// TwinCAT 3 PLC project Plc
// ProgramVersion: 3.1.4024.0
// libraries:
//   Tc2_Standard, * (Beckhoff Automation GmbH)
//   Tc2_System, * (Beckhoff Automation GmbH)
//   Tc2_TcpIp, * (Beckhoff Automation GmbH)
//   Tc3_Module, * (Beckhoff Automation GmbH)
//   VisuSymbols,3.5.10.0,System
// project tree:
//   Elements/Common/ E_Mode.TcDUT, ST_DigitalInput.TcDUT, ST_DigitalOutput.TcDUT, ST_ToggleCmd.TcDUT, ST_TapCmd.TcDUT
//   Elements/Lights/ E_ButtonSelection.TcDUT, FB_AnalogLamp.TcPOU, FB_DigitalLamp.TcPOU, ST_AnalogLamp_cmd.TcDUT, ST_AnalogLamp_fb.TcDUT, ST_DigitalLamp_cmd.TcDUT, ST_DigitalLamp_fb.TcDUT
//   Elements/ ST_AC_Swing.TcDUT, ST_Curtain_Status.TcDUT, ST_ACcontrol.TcDUT, ST_ACStatus.TcDUT, ST_Fan_ip.TcDUT, ST_Fan_op.TcDUT
//   / GlobalTextList.TcGTLO, PlcTask.TcTTO, Visualization Manager.TcVMO (not stored)
//   Helper/ FB_CommandHandling.TcPOU, FB_CurtainPos.TcPOU, F_Scaling.TcPOU (not stored)
//   POUs/ FB_AC.TcPOU, FB_AC_oop.TcPOU, FB_Curtain.TcPOU, FB_Dimmer.TcPOU, FB_Fan.TcPOU, FB_Lamp.TcPOU, FB_Room.TcPOU, I_AC.TcIO, MAIN.TcPOU, PRG_HallRoom.TcPOU, PRG_Kitchen.TcPOU, PRG_SmartHome.TcPOU
//   POUs/TcpIp/ FB_ACcomm.TcPOU, FB_TcpIpClient.TcPOU
//   Trials/ PRG_Testing.TcPOU
//   VISUs/ Template.TcVIS, V_Hall.TcVIS, V_House.TcVIS
// real-time tasks:
//   TASK PlcTask: cycle T#10ms, priority 20, ADS port 350
//   TASK PlcTask1: cycle T#10ms, priority 21, ADS port 351

CONFIGURATION Plc
    RESOURCE PLC ON TwinCAT3
        TASK PlcTask(INTERVAL := T#10ms, PRIORITY := 20);
        PROGRAM MAIN WITH PlcTask : MAIN;
    END_RESOURCE
END_CONFIGURATION

// ---- Elements/Common/E_Mode.TcDUT
{attribute 'qualified_only'}
{attribute 'strict'}
TYPE E_Mode :
(
	auto := 0,
	simulation := 1,
	maintenance := 2,
	manual := 3
);
END_TYPE

// ---- Elements/Common/ST_DigitalInput.TcDUT
TYPE ST_DigitalInput :
STRUCT
	hmi_In: BOOL;
	i_In AT %I* : BOOL;
	mode: E_Mode;
END_STRUCT
END_TYPE

// ---- Elements/Common/ST_DigitalOutput.TcDUT
TYPE ST_DigitalOutput :
STRUCT
	hmi_Out: BOOL;
	q_Out AT %Q* : BOOL;
	mode: E_Mode;
END_STRUCT
END_TYPE

// ---- Elements/Common/ST_ToggleCmd.TcDUT
TYPE ST_ToggleCmd :
STRUCT
	OnOff: BOOL;
END_STRUCT
END_TYPE

// ---- Elements/Common/ST_TapCmd.TcDUT
TYPE ST_TapCmd :
STRUCT
	OnOff: BOOL;
END_STRUCT
END_TYPE

// ---- Elements/Lights/E_ButtonSelection.TcDUT
{attribute 'qualified_only'}
{attribute 'strict'}
TYPE E_ButtonSelection :
(
	Tap := 0,		//	toggle if Event rising edge is detected
	Toggle := 1		//	0: off | 1: on
);
END_TYPE

// ---- Elements/Lights/ST_AnalogLamp_cmd.TcDUT
TYPE ST_AnalogLamp_cmd :
STRUCT
	OnOff: BOOL;
	brightness_SP: INT;	//SP- Setpoint
	colorCode: UDINT;
END_STRUCT
END_TYPE

// ---- Elements/Lights/ST_AnalogLamp_fb.TcDUT
TYPE ST_AnalogLamp_fb :
STRUCT
	status: BOOL;
	brightness: INT;
	colorSelected: UDINT;
	errorID: UDINT;
END_STRUCT
END_TYPE

// ---- Elements/Lights/ST_DigitalLamp_cmd.TcDUT
TYPE ST_DigitalLamp_cmd :
STRUCT
	E_ButtonSelection: E_ButtonSelection;
	Toggle: ST_ToggleCmd;
	PushButton: ST_TapCmd;
END_STRUCT
END_TYPE

// ---- Elements/Lights/ST_DigitalLamp_fb.TcDUT
TYPE ST_DigitalLamp_fb :
STRUCT
	Status: BOOL;
END_STRUCT
END_TYPE

// ---- Elements/ST_AC_Swing.TcDUT
TYPE ST_AC_Swing :
STRUCT
	HorizOn: BOOL;
	HorizOff: BOOL;
	VertiOn: BOOL;
	VertiOff: BOOL;
END_STRUCT
END_TYPE

// ---- Elements/ST_Curtain_Status.TcDUT
TYPE ST_Curtain_Status :
STRUCT
	Open	  	: BOOL;
	Close	 	: BOOL;
	OpenPerc	: INT; 	//0: Closed .. 100: Full Open	
	OpenToCloseTime: TIME := T#10S;
END_STRUCT
END_TYPE

// ---- Elements/ST_ACcontrol.TcDUT
TYPE ST_ACcontrol :
STRUCT
	OnCmd: BOOL;
	OffCmd: BOOL;
	modeSelection: INT;
	swing: ST_AC_Swing;
	tempUp: BOOL;
	tempDown: BOOL;
	tempSP: REAL;
	tempSP_prev: REAL;
END_STRUCT
END_TYPE

// ---- Elements/ST_ACStatus.TcDUT
TYPE ST_ACStatus :
STRUCT
	OnOff: BOOL;
	mode: INT;
	HorizSwingOnOff: BOOL;
	VertiSwingOnOff: BOOL;
	temp: REAL;
END_STRUCT
END_TYPE

// ---- Elements/ST_Fan_ip.TcDUT
TYPE ST_Fan_ip :
STRUCT
	OnOffCmd 	AT%I* : BOOL;
	SpeedSp		AT%I* : INT;
END_STRUCT
END_TYPE

// ---- Elements/ST_Fan_op.TcDUT
TYPE ST_Fan_op :
STRUCT
	OnOff	 	AT%Q* : BOOL;
	Speed		AT%Q* : INT;
END_STRUCT
END_TYPE

// ---- POUs/I_AC.TcIO
INTERFACE I_AC

PROPERTY AC_IPAddr : STRING
GET
END_GET
END_PROPERTY

PROPERTY ACcontrol : ST_ACcontrol
GET
END_GET
END_PROPERTY

PROPERTY ACstatus : ST_ACStatus
SET
END_SET
END_PROPERTY

END_INTERFACE

// ---- POUs/MAIN.TcPOU
PROGRAM MAIN
VAR
END_VAR


	PRG_SmartHome();
	PRG_Testing();

END_PROGRAM

// ---- POUs/PRG_SmartHome.TcPOU
PROGRAM PRG_SmartHome
VAR
	fbRoom: ARRAY[0..1] OF FB_Room;
	AC_IPAddr: STRING := '192.168.1.7';
END_VAR


	fbRoom[0](AC_IPAddr := AC_IPAddr, ACcontrol:= , ACstatus=> );
//	fbRoom[1](AC_IPAddr := );
//	PRG_HallRoom();
//	PRG_Kitchen();

END_PROGRAM

// ---- POUs/FB_Room.TcPOU
FUNCTION_BLOCK FB_Room
VAR_INPUT
	AC_IPAddr: STRING;
	ACcontrol: ST_ACcontrol;
END_VAR
VAR_OUTPUT
	ACstatus: ST_ACStatus;
END_VAR
VAR
	fbLamp : ARRAY[0..3] OF FB_Lamp;
	fbDimmer : ARRAY[0..3] OF FB_Dimmer;
	fbCurtain: FB_Curtain;
	fbAC: FB_AC;
	i: INT;
	fbAC_oop: FB_AC_oop;
END_VAR

	
	FOR i := 0 TO 3 BY 1 DO
		fbLamp[i]();
		fbDimmer[i]();
	END_FOR
	
	//fbAC(AC_IPAddr	:=	AC_IPAddr, ACcontrol:= ACcontrol, ACstatus=> ACstatus);
	fbCurtain();

END_FUNCTION_BLOCK

// ---- POUs/FB_Lamp.TcPOU
FUNCTION_BLOCK FB_Lamp
VAR_INPUT
END_VAR
VAR_OUTPUT
END_VAR
VAR
	Key				AT %I* 	: BOOL;
	Lamp			AT %Q* 	: BOOL;
	rtKey: R_TRIG;
END_VAR


	rtKey(CLK:= Key, Q=> );
	IF rtKey.Q THEN
		Lamp		:=	NOT Lamp;
	END_IF

END_FUNCTION_BLOCK

// ---- POUs/FB_Dimmer.TcPOU
FUNCTION_BLOCK FB_Dimmer
VAR_INPUT
END_VAR
VAR_OUTPUT
END_VAR
VAR
	rotarySw		AT %I* 	: INT;
	Dimmer			AT %Q* 	: INT;
END_VAR


	Dimmer	:=	REAL_TO_INT(F_Scaling(Variable_In:= rotarySw, ZeroIn:= 0, ZeroOut:= 100, SpanIn:= -32768, SpanOut:= 32767));

END_FUNCTION_BLOCK

// ---- POUs/FB_Curtain.TcPOU
FUNCTION_BLOCK FB_Curtain
VAR_INPUT
END_VAR
VAR_OUTPUT
END_VAR
VAR
	OpenCmd AT%I* : BOOL;
	CloseCmd AT%I* : BOOL;	
	AtOpen	 AT%I* 	: BOOL;		// Sensor Feedback	
	AtClose	 AT%I*	: BOOL;		// Sensor Feedback

	Open	 AT%Q* : BOOL;
	Close	 AT%Q* : BOOL;	
	
	OpenPerc	: INT; 	//0: Closed .. 100: Full Open	
	OpenToCloseTime: INT := 10000;	
	fbCurtainPos: FB_CurtainPos;
	rtOpenCmd: R_TRIG;
	rtCloseCmd: R_TRIG;
END_VAR


	rtOpenCmd(CLK:= OpenCmd, Q=> );
	rtCloseCmd(CLK:= CloseCmd, Q=> );
	
	IF rtOpenCmd.Q THEN
		Open		:=	NOT Open;
		Close		:=	FALSE;
	END_IF
	IF rtCloseCmd.Q THEN
		Open		:=	FALSE;
		Close		:=	NOT Close;
	END_IF
	
	IF AtOpen THEN
		Open		:=	FALSE;
	END_IF
	IF AtClose THEN
		Close		:=	FALSE;
	END_IF
	
	fbCurtainPos(
		OpenCmd:= Open,
		CloseCmd:= Close,
		AtOpen:= AtOpen, 
		AtClose:= AtClose, 
		plcCylTime_mSec:= 10, 
		OpenToCloseTime:= OpenToCloseTime, 
		OpenPerc=> OpenPerc);

END_FUNCTION_BLOCK

// ---- Helper/FB_CurtainPos.TcPOU
FUNCTION_BLOCK FB_CurtainPos
VAR_INPUT
	OpenCmd: BOOL;
	CloseCmd: BOOL;
	AtOpen: BOOL;
	AtClose: BOOL;
	plcCylTime_mSec: INT := 10;
	OpenToCloseTime: INT;
END_VAR
VAR_OUTPUT
	OpenPerc: INT;
END_VAR
VAR
	rtAtOpen : R_TRIG;
	rtAtClose : R_TRIG;
	OpenPerc_Loc: INT;
END_VAR


	rtAtOpen(CLK:= AtOpen, Q=> );
	rtAtClose(CLK:= AtClose, Q=> );
	
	IF rtAtOpen.Q THEN
		OpenPerc		:=	100;
	END_IF
	IF rtAtClose.Q THEN
		OpenPerc		:=	0;
	END_IF
	
	IF (OpenCmd) THEN
		OpenPerc_Loc	:=	LIMIT(0 , OpenPerc_Loc + plcCylTime_mSec, OpenToCloseTime);
		OpenPerc		:=	(REAL_TO_INT(F_Scaling(Variable_In:= OpenPerc_Loc, ZeroIn:= 0, ZeroOut:= OpenToCloseTime, SpanIn:= 0, SpanOut:= 100)));
	END_IF

	IF (CloseCmd) THEN
		OpenPerc_Loc	:=	LIMIT(0 , OpenPerc_Loc - plcCylTime_mSec, OpenToCloseTime);
		OpenPerc		:=	(REAL_TO_INT(F_Scaling(Variable_In:= OpenPerc_Loc, ZeroIn:= 0, ZeroOut:= OpenToCloseTime, SpanIn:= 0, SpanOut:= 100)));
	END_IF

END_FUNCTION_BLOCK

// ---- POUs/FB_AC.TcPOU
FUNCTION_BLOCK FB_AC
VAR_INPUT
	AC_IPAddr: STRING;
	ACcontrol: ST_ACcontrol;
END_VAR
VAR_OUTPUT
	ACstatus: ST_ACStatus;
END_VAR
VAR
	fbACcomm: FB_ACcomm;
	prevMode: INT;
	step: (eIdle, eOn, eOff, eModeChange, eError);
	fbOnCmd: FB_CommandHandling;
	fbOffCmd: FB_CommandHandling;
	fbModeChangeCmd: FB_CommandHandling;
END_VAR

VAR CONSTANT
	cOnCmd: STRING := 'AC On Cmd';
	cOffCmd: STRING := 'AC Off Cmd';
	cModeChangeCmd: STRING := 'AC Mode = ';
END_VAR


	fbACcomm( AC_IPAddr	:=	AC_IPAddr );
	
	fbOnCmd(cmd:= ACcontrol.OnCmd, timeoutOccured => , reset:= , timeout:= , Q=> );
	fbOffCmd(cmd:= ACcontrol.OffCmd, timeoutOccured => , reset:= , timeout:= , Q=> );
	fbModeChangeCmd(cmd:= ACcontrol.modeSelection <> prevMode, timeoutOccured => , reset:= , timeout:= , Q=> );
	prevMode	:=	ACcontrol.modeSelection;
	
	CASE step OF 
	eIdle: 
		IF fbOnCmd.Q THEN
			step		:=	eOn;
		END_IF
		IF fbOffCmd.Q THEN
			step		:=	eOff;
		END_IF
		IF fbModeChangeCmd.Q THEN
			step		:=	eModeChange;
		END_IF
			
	eOn:
		fbACcomm(sCmd:= cOnCmd, bSend:= TRUE);
		IF fbACcomm.bResponseReceived OR fbACcomm.bNoResponse THEN
			fbACcomm(sCmd:= , bSend:= FALSE );
			step		:=	eIdle;
		END_IF
		
	eOff:
		fbACcomm(sCmd:= cOffCmd, bSend:= TRUE);
		IF fbACcomm.bResponseReceived OR fbACcomm.bNoResponse THEN
			fbACcomm(sCmd:= , bSend:= FALSE );
			step		:=	eIdle;
		END_IF
		
	eModeChange:
		fbACcomm(sCmd:= CONCAT(cModeChangeCmd, INT_TO_STRING(ACcontrol.modeSelection)), bSend:= TRUE);
		IF fbACcomm.bResponseReceived OR fbACcomm.bNoResponse THEN
			fbACcomm(sCmd:= , bSend:= FALSE );
			step		:=	eIdle;
		END_IF
		
	eError:
	END_CASE

END_FUNCTION_BLOCK

// ---- POUs/TcpIp/FB_ACcomm.TcPOU
FUNCTION_BLOCK FB_ACcomm
VAR_INPUT
	AC_IPAddr: STRING;
	sCmd: STRING;
	bSend: BOOL;
END_VAR
VAR_OUTPUT
	sResponse: STRING;
	bResponseReceived: BOOL;
	bNoResponse: BOOL;
END_VAR
VAR
	fbTcpIpCommWithAC: FB_TcpIpClient;
	step_ACcomm: (eIdle, eError, ePreConnect, eConnect, eMonitor, eOn, eOff, eModeChange, eSwing, eTempChange);
	
	rtSend: R_TRIG;
	tonSendCmdTimeout: TON;
	fbSendCmd: FB_CommandHandling;
END_VAR


	fbSendCmd(cmd:= bSend, reset:= fbTcpIpCommWithAC.bSendSuccess, timeoutOccured => bNoResponse, timeout:= , Q=> );
	
	CASE step_ACcomm OF
	eIdle:
		IF (fbTcpIpCommWithAC.srvIpAddr <> '') AND (NOT fbTcpIpCommWithAC.connected) AND (NOT fbTcpIpCommWithAC.busy) THEN
			fbTcpIpCommWithAC(connect:= FALSE);
			step_ACcomm		:=	ePreConnect;
		END_IF
		
	ePreConnect: 
		fbTcpIpCommWithAC(
			connect			:= TRUE, 
			srvIpAddr		:= AC_IPAddr, 
			port			:= 23);
		
		IF fbTcpIpCommWithAC.busy THEN
			step_ACcomm		:=	eMonitor;
		ELSIF fbTcpIpCommWithAC.errId <> 0 THEN
			step_ACcomm		:=	eError;
		END_IF
			
	eConnect:
		fbTcpIpCommWithAC(
			connect			:= FALSE, 
			srvIpAddr		:= AC_IPAddr, 
			port			:= 23);
		
		IF (NOT fbTcpIpCommWithAC.busy) AND (fbTcpIpCommWithAC.connected) THEN
			step_ACcomm		:=	eMonitor;
		ELSIF fbTcpIpCommWithAC.errId <> 0 THEN
			step_ACcomm		:=	eError;
		END_IF
					
	eMonitor:
		fbTcpIpCommWithAC(sData	:=	sCmd, send:= fbSendCmd.Q, sReceivedData => sResponse);
	
		IF fbTcpIpCommWithAC.errId <> 0 THEN
			step_ACcomm		:=	eError;	
		END_IF
		
	eError:	
		step_ACcomm			:=	eIdle;
	END_CASE
	
	fbTcpIpCommWithAC(
		connect:= , 
		srvIpAddr:= AC_IPAddr, 
		port:= , 
		sData:= , 
		send:= , 
		reset:= , 
		close:= , 
		closeAll:= , 
		busy=> , 
		connected=> , 
		bSendSuccess => ,
		sReceivedData=> , 
		nRecBytes=> , 
		bRecSuccess => bResponseReceived,
		errId=> );

END_FUNCTION_BLOCK

// ---- POUs/TcpIp/FB_TcpIpClient.TcPOU
FUNCTION_BLOCK FB_TcpIpClient
VAR_INPUT
	connect: BOOL;
	srvIpAddr: STRING;	//Server's IP Address
	port: UDINT;
	sData: STRING(255);
	send: BOOL;
	reset: BOOL;
	close: BOOL;
	closeAll: BOOL;
END_VAR
VAR_OUTPUT
	busy: BOOL;
	connected: BOOL;
	bSendSuccess: BOOL;
	sReceivedData: STRING(255);
	nRecBytes: UDINT;
	bRecSuccess: BOOL;
	errId: UDINT;
END_VAR
VAR
	fbConnect: FB_SocketConnect;
	fbClose: FB_SocketClose;
	fbCloseAll: FB_SocketCloseAll;
	fbSend: FB_SocketSend;
	fbReceive: FB_SocketReceive;
	step: (eIdle, eInit, eError, ePreConnect, eConnect, ePreClose, eClose, ePreCloseAll, eCloseAll, ePreSend, eSend);
	step_rec: (eIdle_rec, ePreReceive_rec, eReceive_rec, eWait_rec, eError_rec);
	rtConnect: R_TRIG;
	rtClose: R_TRIG;
	rtCloseAll: R_TRIG;
	rtReset: R_TRIG;
	rtSend: R_TRIG;
	tonWait: TON;
	sReceivedData_loc: STRING(255);	
	M_ErrGeneratedAtRec: BOOL;
END_VAR

VAR CONSTANT
	NullChar: BYTE := 0;
END_VAR

	rtConnect	(CLK:= connect, Q=> );
	rtClose		(CLK:= close, Q=> );
	rtCloseAll	(CLK:= closeAll, Q=> );	
	rtReset		(CLK:= reset, Q=> );	
	rtSend		(CLK:= send, Q=> );	

	IF bSendSuccess AND (NOT send) THEN
		bSendSuccess			:=	FALSE;
	END_IF
	
	CASE step OF
	eIdle:			
		IF rtConnect.Q THEN
			errId				:=	0;
			busy				:=	TRUE;
			connected			:=	FALSE;
			step				:=	eInit;
		END_IF
		IF rtClose.Q THEN
			fbClose(bExecute	:= FALSE);
			errId				:=	0;
			busy				:=	TRUE;
			step				:=	ePreClose;			
		END_IF
		IF rtCloseAll.Q THEN
			fbCloseAll(	bExecute:= FALSE);
			errId				:=	0; 
			busy				:=	TRUE;
			step				:=	ePreCloseAll;
		END_IF
		IF rtSend.Q THEN
			fbSend(bExecute		:=	FALSE);
			busy				:=	TRUE;
			errId				:=	0;
			step				:=	ePreSend;
		END_IF

	eInit:
	
		fbConnect(
			sSrvNetId		:= '', 
			sRemoteHost		:= srvIpAddr, 
			nRemotePort		:= port, 
			bExecute		:= FALSE, 
			tTimeout		:= DEFAULT_ADS_TIMEOUT, 
			bBusy			=> , 
			bError			=> , 
			nErrId			=> , 
			hSocket			=> );

		fbClose(
			sSrvNetId		:= '', 
			hSocket			:= fbConnect.hSocket, 
			bExecute		:= FALSE, 
			tTimeout		:= DEFAULT_ADS_TIMEOUT, 
			bBusy			=> , 
			bError			=> , 
			nErrId			=> );
			
		fbCloseAll(
			sSrvNetId		:= '', 
			bExecute		:= FALSE, 
			tTimeout		:= DEFAULT_ADS_TIMEOUT, 
			bBusy			=> , 
			bError			=> , 
			nErrId			=> );
			
		fbSend(
			sSrvNetId		:= '', 
			hSocket			:= , 
			cbLen			:= , 
			pSrc			:= , 
			bExecute		:= FALSE, 
			tTimeout		:= DEFAULT_ADS_TIMEOUT, 
			bBusy			=> , 
			bError			=> , 
			nErrId			=> );
			
		step				:=	ePreConnect;
		
	ePreConnect:
		fbConnect(
			bExecute		:= TRUE, 
			tTimeout		:= DEFAULT_ADS_TIMEOUT,  
			hSocket			=> );	
			
		IF fbConnect.bBusy THEN
			step			:=	eConnect;
		ELSIF fbConnect.bError THEN
			errID			:=	fbConnect.nErrId;
			step			:=	eError;	
		END_IF
	
	eConnect:	
		fbConnect(
			bExecute		:= FALSE, 
			tTimeout		:= DEFAULT_ADS_TIMEOUT,  
			hSocket			=> );	
			
		IF (NOT fbConnect.bBusy) AND (NOT fbConnect.bError) AND (fbConnect.hSocket.handle <> 0) THEN
			connected		:=	TRUE;
			busy			:=	FALSE;
			step			:=	eIdle;
		ELSIF fbConnect.bError THEN
			errID			:=	fbConnect.nErrId;
			step			:=	eError;	
		END_IF
		
	ePreClose:
		fbClose(
			hSocket			:= fbConnect.hSocket, 
			bExecute		:= TRUE);
			
		IF fbClose.bBusy THEN
			step			:=	eClose;
		ELSIF fbCLose.bError THEN
			errID			:=	fbClose.nErrId;
			step			:=	eError;
		END_IF
	
	eClose:
		fbClose(
			hSocket			:= fbConnect.hSocket, 
			bExecute		:= FALSE);
			
		IF (NOT fbClose.bBusy) AND (NOT fbClose.bError) THEN
			step			:=	eIdle;
			connected		:=	FALSE;
			busy			:=	FALSE;
		ELSIF fbCLose.bError THEN
			errID			:=	fbClose.nErrId;
			step			:=	eError;
		END_IF
		
	ePreCloseAll:
		fbCloseAll(bExecute		:= TRUE);
			
		IF fbCloseAll.bBusy THEN
			step			:=	eCloseAll;
		ELSIF fbCloseAll.bError THEN
			errID			:=	fbCloseAll.nErrId;
			step			:=	eError;
		END_IF
	
	eCloseAll:
		fbCloseAll(bExecute		:= FALSE);
			
		IF (NOT fbCloseAll.bBusy) AND (NOT fbCloseAll.bError) THEN
			step			:=	eIdle;
			connected		:=	FALSE;
			busy			:=	FALSE;
		ELSIF fbCloseAll.bError THEN
			errID			:=	fbCloseAll.nErrId;
			step			:=	eError;
		END_IF
	
	ePreSend:
		fbSend( 
			hSocket			:= fbConnect.hSocket, 
			cbLen			:= LEN(sData), 
			pSrc			:= ADR(sData), 
			bExecute		:= TRUE);

		IF (fbSend.bBusy) THEN
			step			:=	eSend;
		ELSIF fbSend.bError THEN
			errID			:=	fbSend.nErrId;
			step			:=	eError;
		END_IF
	
	eSend:
		fbSend( 
			hSocket			:= fbConnect.hSocket, 
			cbLen			:= LEN(sData), 
			pSrc			:= ADR(sData), 
			bExecute		:= FALSE);

		IF (NOT fbSend.bBusy) AND (NOT fbSend.bError) THEN
			bSendSuccess	:=	TRUE;
			busy			:=	FALSE;
			step			:=	eIdle;
		ELSIF fbSend.bError THEN
			errID			:=	fbSend.nErrId;
			step			:=	eError;
		END_IF
		
	eError:
		busy				:=	FALSE;
		
		step				:=	eIdle;
//		IF rtReset.Q THEN
//			step			:=	eIdle;
//			errID			:=	0;
//		END_IF
		
	END_CASE
	
//	################################
	CASE step_rec OF
	eIdle_rec:
		IF connected THEN
			fbReceive(
				sSrvNetId		:= '', 
				hSocket			:= fbConnect.hSocket, 
				bExecute		:= FALSE, 
				tTimeout		:= DEFAULT_ADS_TIMEOUT, 
				bBusy			=> , 
				bError			=> , 
				nErrId			=> , 
				nRecBytes		=> nRecBytes);
			
			//MEMCPY(destAddr:= ADR(sReceivedData_loc), srcAddr:= ADR(NullChar), n:= SIZEOF(sReceivedData_loc));	
			tonWait(IN:= FALSE);
			step_rec			:=	ePreReceive_rec;	
		END_IF
		bRecSuccess				:=	FALSE;
		
	ePreReceive_rec:
		fbReceive( 
			cbLen			:= SIZEOF(sReceivedData_loc), 
			pDest			:= ADR(sReceivedData_loc), 
			bExecute		:= TRUE, 
			nRecBytes		=> nRecBytes);	
		
		IF fbReceive.bBusy THEN
			step_rec		:=	eReceive_rec;
		ELSIF fbReceive.bError THEN
			errId			:=	fbReceive.nErrId;
			M_ErrGeneratedAtRec	:=	TRUE;
			step_rec		:=	eError_rec;			
		END_IF
	
	eReceive_rec:
		fbReceive( 
			cbLen			:= SIZEOF(sReceivedData_loc), 
			pDest			:= ADR(sReceivedData_loc), 
			bExecute		:= FALSE, 
			nRecBytes		=> nRecBytes);	
		
		IF (NOT fbReceive.bBusy) AND (NOT fbReceive.bError) THEN			
			IF nRecBytes > 0 THEN				
				sReceivedData		:=	LEFT(sReceivedData_loc, UDINT_TO_INT(nRecBytes));
				bRecSuccess			:=	TRUE;
			END_IF
			step_rec		:=	eWait_rec;			
		ELSIF fbReceive.bError THEN
			errId			:=	fbReceive.nErrId;
			M_ErrGeneratedAtRec	:=	TRUE;
			step_rec		:=	eError_rec;
		END_IF	
			
	eWait_rec:
		tonWait(IN:= TRUE, PT:= T#2S, Q=> , ET=> );
		IF tonWait.Q THEN
			step_rec			:=	eIdle_rec;
			tonWait(IN:= FALSE);
		END_IF
		
	eError_rec:
		tonWait(IN:= TRUE, PT:= T#2S, Q=> , ET=> );
		
		fbReceive(
			bExecute		:= FALSE);
			
		IF tonWait.Q THEN
			IF M_ErrGeneratedAtRec THEN
				errId					:=	0;
				M_ErrGeneratedAtRec		:=	FALSE;
			END_IF			
			tonWait(IN:= FALSE);
			step_rec			:=	eIdle_rec;			
		END_IF
		
	END_CASE
	
//	Calling	############################
	fbConnect(
		sSrvNetId		:= , 
		sRemoteHost		:= , 
		nRemotePort		:= , 
		bExecute		:= , 
		tTimeout		:= , 
		bBusy			=> , 
		bError			=> , 
		nErrId			=> , 
		hSocket			=> );
		
	fbClose(
		sSrvNetId		:= , 
		hSocket			:= , 
		bExecute		:= , 
		tTimeout		:= , 
		bBusy			=> , 
		bError			=> , 
		nErrId			=> );
		
	fbCloseAll(
		sSrvNetId		:= , 
		bExecute		:= , 
		tTimeout		:= , 
		bBusy			=> , 
		bError			=> , 
		nErrId			=> );
		
	fbSend(
		sSrvNetId		:= , 
		hSocket			:= , 
		cbLen			:= , 
		pSrc			:= , 
		bExecute		:= , 
		tTimeout		:= , 
		bBusy			=> , 
		bError			=> , 
		nErrId			=> );

	fbReceive(
		sSrvNetId		:= , 
		hSocket			:= , 
		cbLen			:= , 
		pDest			:= , 
		bExecute		:= , 
		tTimeout		:= , 
		bBusy			=> , 
		bError			=> , 
		nErrId			=> , 
		nRecBytes		=> );

END_FUNCTION_BLOCK

// ---- Helper/FB_CommandHandling.TcPOU
FUNCTION_BLOCK FB_CommandHandling
VAR_INPUT
	cmd: BOOL;
	reset: BOOL;
	timeout: INT := 5000;		//	in mSec
END_VAR
VAR_OUTPUT
	Q: BOOL;
	timeoutOccured: BOOL;
END_VAR
VAR
	tonTimeout: TON;
	rtCmd: R_TRIG;
	rtReset: R_TRIG;
END_VAR

	rtCmd(CLK:= cmd, Q=> );
	rtReset(CLK:= reset, Q=> );

	IF rtCmd.Q THEN
		Q				:=	TRUE;
		timeoutOccured	:=	FALSE;
	END_IF
	IF NOT cmd THEN
		Q				:=	FALSE;
		timeoutOccured	:=	FALSE;		
	END_IF
	tonTimeout(IN:= cmd, PT:= INT_TO_TIME(timeout), Q=> , ET=> );
	IF tonTimeout.Q THEN
		Q				:=	FALSE;
		timeoutOccured	:=	TRUE;
	END_IF
	IF rtReset.Q THEN
		Q				:=	FALSE;
	END_IF

END_FUNCTION_BLOCK

// ---- POUs/FB_AC_oop.TcPOU
FUNCTION_BLOCK FB_AC_oop IMPLEMENTS I_AC
VAR_INPUT
//	AC_IPAddr: STRING;
//	ACcontrol: ST_ACcontrol;
END_VAR
VAR_OUTPUT
//	ACstatus: ST_ACStatus;
END_VAR
VAR
	_AC_IPAddr: STRING;
	_ACcontrol: ST_ACcontrol;
	_ACstatus: ST_ACStatus;	
	
	fbACcomm: FB_ACcomm;
	prevMode: INT;
	step: (eIdle, eOn, eOff, eModeChange, eError);
	fbOnCmd: FB_CommandHandling;
	fbOffCmd: FB_CommandHandling;
	fbModeChangeCmd: FB_CommandHandling;
END_VAR

VAR CONSTANT
	cOnCmd: STRING := 'AC On Cmd';
	cOffCmd: STRING := 'AC Off Cmd';
	cModeChangeCmd: STRING := 'AC Mode = ';
END_VAR


	fbACcomm( AC_IPAddr	:=	AC_IPAddr );
	
	fbOnCmd(cmd:= _ACcontrol.OnCmd, timeoutOccured => , reset:= , timeout:= , Q=> );
	fbOffCmd(cmd:= _ACcontrol.OffCmd, timeoutOccured => , reset:= , timeout:= , Q=> );
	fbModeChangeCmd(cmd:= _ACcontrol.modeSelection <> prevMode, timeoutOccured => , reset:= , timeout:= , Q=> );
	prevMode	:=	_ACcontrol.modeSelection;
	
	CASE step OF 
	eIdle: 
		IF fbOnCmd.Q THEN
			step		:=	eOn;
		END_IF
		IF fbOffCmd.Q THEN
			step		:=	eOff;
		END_IF
		IF fbModeChangeCmd.Q THEN
			step		:=	eModeChange;
		END_IF
			
	eOn:
		fbACcomm(sCmd:= cOnCmd, bSend:= TRUE);
		IF fbACcomm.bResponseReceived OR fbACcomm.bNoResponse THEN
			fbACcomm(sCmd:= , bSend:= FALSE );
			step		:=	eIdle;
		END_IF
		
	eOff:
		fbACcomm(sCmd:= cOffCmd, bSend:= TRUE);
		IF fbACcomm.bResponseReceived OR fbACcomm.bNoResponse THEN
			fbACcomm(sCmd:= , bSend:= FALSE );
			step		:=	eIdle;
		END_IF
		
	eModeChange:
		fbACcomm(sCmd:= CONCAT(cModeChangeCmd, INT_TO_STRING(_ACcontrol.modeSelection)), bSend:= TRUE);
		IF fbACcomm.bResponseReceived OR fbACcomm.bNoResponse THEN
			fbACcomm(sCmd:= , bSend:= FALSE );
			step		:=	eIdle;
		END_IF
		
	eError:
	END_CASE

{warning 'add property implementation'}
PROPERTY AC_IPAddr : STRING
GET
_AC_IPAddr	:=	AC_IPAddr;
END_GET
END_PROPERTY

{warning 'add property implementation'}
PROPERTY ACcontrol : ST_ACcontrol
GET
_ACcontrol	:=	ACcontrol;
END_GET
END_PROPERTY

{warning 'add property implementation'}
PROPERTY ACstatus : ST_ACStatus
SET
ACstatus	:=	_ACstatus;
END_SET
END_PROPERTY

END_FUNCTION_BLOCK

// ---- Trials/PRG_Testing.TcPOU
PROGRAM PRG_Testing
VAR
	fbTcpIpClient: FB_TcpIpClient;
	connect: BOOL;
	reset: BOOL;
	close: BOOL;
	closeAll: BOOL;
	busy: BOOL;
	connected: BOOL;
	errId: UDINT;
	sData: STRING(255);
	send: BOOL;
	sReceivedData: STRING(255);
	nRecBytes: UDINT;
END_VAR


	fbTcpIpClient(
		connect:= connect, 
		srvIpAddr:= '192.168.1.7', 
		port:= 23, 
		sData:= sData,
		send:= send,
		reset:= reset, 
		close:= close, 
		closeAll:= closeAll, 
		busy=> busy, 
		connected=> connected, 
		bSendSuccess => ,		
		sReceivedData=> sReceivedData,
		nRecBytes=> nRecBytes,
		bRecSuccess => ,
		errId=> errId);

	connect	:=	FALSE;
	reset	:=	FALSE;
	close	:=	FALSE;
	closeAll	:=	FALSE;
	send:=	FALSE;

END_PROGRAM

// ---- Elements/Lights/FB_AnalogLamp.TcPOU
FUNCTION_BLOCK FB_AnalogLamp
VAR_INPUT
END_VAR
VAR_OUTPUT
END_VAR
VAR
END_VAR

END_FUNCTION_BLOCK

// ---- Elements/Lights/FB_DigitalLamp.TcPOU
FUNCTION_BLOCK FB_DigitalLamp
VAR_INPUT
	Lamp_cmd: ST_DigitalLamp_cmd;
END_VAR
VAR_OUTPUT
	Lamp_fb: ST_DigitalLamp_fb;
END_VAR
VAR
	rtOnOff_PushButton: R_TRIG;	
END_VAR


	rtOnOff_PushButton(CLK:= Lamp_cmd.PushButton, Q=> );
	
	IF Lamp_cmd.E_ButtonSelection = E_ButtonSelection.Toggle THEN
		IF Lamp_cmd.Toggle.OnOff THEN
			Lamp_fb.Status	:=	TRUE;
		END_IF
		IF NOT Lamp_cmd.Toggle.OnOff THEN
			Lamp_fb.Status	:=	FALSE;
		END_IF
	ELSIF Lamp_cmd.E_ButtonSelection = E_ButtonSelection.Tap THEN
		IF rtOnOff_PushButton.Q THEN
			Lamp_fb.Status	:=	NOT Lamp_fb.Status;
		END_IF
	ELSE
		Lamp_fb.Status		:=	FALSE;
	END_IF

END_FUNCTION_BLOCK

// ---- POUs/FB_Fan.TcPOU
FUNCTION_BLOCK FB_Fan
VAR_INPUT
END_VAR
VAR_OUTPUT
END_VAR
VAR
	FanControl				: ST_Fan_ip;
	Fan						: ST_Fan_op;
	rtFanOnOffCmd: R_TRIG;
END_VAR


	rtFanOnOffCmd(CLK:= FanControl.OnOffCmd, Q=> );
	IF rtFanOnOffCmd.Q THEN
		Fan.OnOff		:=	NOT Fan.OnOff;
	END_IF
	Fan.Speed			:=	FanControl.SpeedSp;

END_FUNCTION_BLOCK

// ---- POUs/PRG_HallRoom.TcPOU
PROGRAM PRG_HallRoom
VAR
	fbLamp : ARRAY[0..3] OF FB_Lamp;
	fbDimmer : ARRAY[0..3] OF FB_Dimmer;
	fbFan: FB_Fan;
	fbCurtain: FB_Curtain;
	i: INT;	
END_VAR


	FOR i := 0 TO 3 BY 1 DO
		fbLamp[i]();
		fbDimmer[i]();
	END_FOR
	fbFan();
	
	fbCurtain();

END_PROGRAM

// ---- POUs/PRG_Kitchen.TcPOU
PROGRAM PRG_Kitchen
VAR
	fbLamp : ARRAY[0..1] OF FB_Lamp;
	fbDimmer : ARRAY[0..1] OF FB_Dimmer;
	i: INT;	
END_VAR


	FOR i := 0 TO 1 BY 1 DO
		fbLamp[i]();
		fbDimmer[i]();
	END_FOR

END_PROGRAM

// ---- GlobalTextList.TcGTLO
TEXTLIST GlobalTextList
  974 = '%i'
  712 = '1'
  147 = '2'
  377 = '3'
  67 = '4'
  437 = '5'
  273 = '6'
  894 = '7'
  89 = '8'
  35 = 'Bedroom 1'
  598 = 'Bedroom 2'
  112 = 'Hall'
  506 = 'Kitchen'
  393 = 'Sweet Home'
END_TEXTLIST

// ---- VISUs/Template.TcVIS
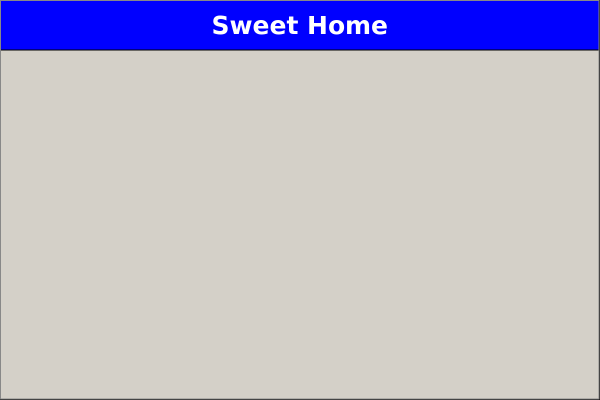
VISUALIZATION Template  // 600x400
    Rectangle (0,0 600x400)
    Rectangle (0,0 600x50), "Sweet Home"
END_VISUALIZATION

// ---- VISUs/V_Hall.TcVIS
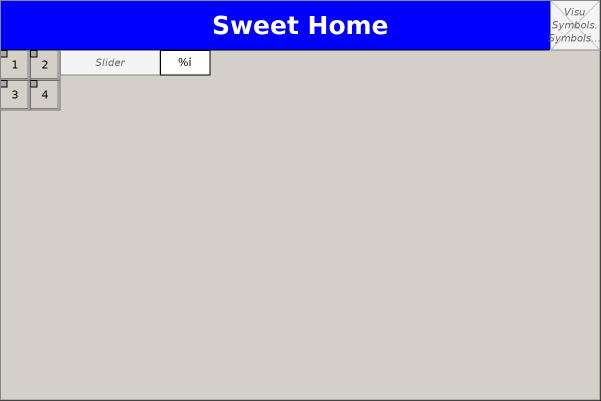
VISUALIZATION V_Hall  // 601x401
    Frame (0,0 601x401)
        shows Template()
    Image (550,0 50x50), image: VisuSymbols.Symbols.Home
        OnMouseClick: change screen: V_House
    Button (0,50 30x30), "1"
        tap PRG_SmartHome.fbRoom.fbLamp[0].Key
    Rectangle (0,50 7x7), colour toggle: PRG_SmartHome.fbRoom.fbLamp[0].Lamp
    Button (30,50 30x30), "2"
        tap PRG_SmartHome.fbRoom.fbLamp[1].Key
    Rectangle (30,50 7x7), colour toggle: PRG_SmartHome.fbRoom.fbLamp[1].Lamp
    Button (30,80 30x30), "4"
        tap PRG_SmartHome.fbRoom.fbLamp[3].Key
    Rectangle (30,80 7x7), colour toggle: PRG_SmartHome.fbRoom.fbLamp[3].Lamp
    Button (0,80 30x30), "3"
        tap PRG_SmartHome.fbRoom.fbLamp[2].Key
    Rectangle (0,80 7x7), colour toggle: PRG_SmartHome.fbRoom.fbLamp[2].Lamp
    Slider (60,50 100x25), variable: PRG_SmartHome.fbRoom.fbDimmer[0].rotarySw, scale 0..100
    Rectangle (160,50 50x25), "%i", text variable: PRG_SmartHome.fbRoom.fbDimmer[0].Dimmer
END_VISUALIZATION

// ---- VISUs/V_House.TcVIS
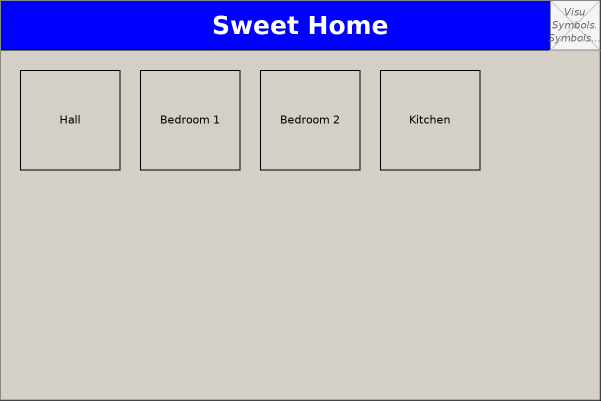
VISUALIZATION V_House  // 601x401
    Frame (0,0 601x401)
        shows Template()
    Rectangle (20,70 100x100), "Hall"
        OnMouseClick: change screen: V_Hall
    Rectangle (140,70 100x100), "Bedroom 1"
    Rectangle (260,70 100x100), "Bedroom 2"
    Rectangle (380,70 100x100), "Kitchen"
    Image (550,0 50x50), image: VisuSymbols.Symbols.Home
        OnMouseClick: change screen: V_House
END_VISUALIZATION
